Universal Robots PolyScope program: Albert_Miquel.urp

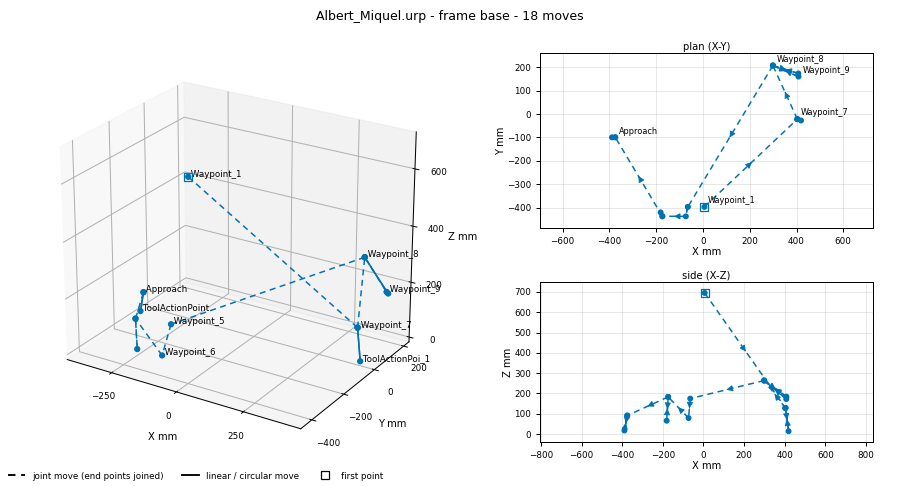
[picture p0: tool path of Albert_Miquel.urp in frame base, 18 of 18 moves have a stored position in this frame; points joined in program order, loops and branches not executed]
Program Albert_Miquel (installation=default directory=/programs createdIn=5.14.5 lastSavedIn=5.14.5 robotSerialNumber=20195300809)
Calibrated DH parameters: a=[-0.000085, -0.20076, -0.212369, 0.000121, -0.000118, 0]; d=[0.15185, -26.306375, 24.753047, 1.684739, 0.085386, 0.092088]; alpha=[1.572149, -0.00522, -0.011864, 1.571339, -1.571085, 0]; deltaTheta=[0, 0.599885, -0.513355, -0.086555, 0.000006, 0]
InitVariablesNode variables(variable(name=Pallet_1_cnt_1, expression=1), variable(name=Pallet_1_cnt_2, expression=1), variable(name=Pallet_1_lct_1, expression=1), variable(name=Pallet_1_lct_2, expression=1), variable(name=Pallet_1_lno_1, expression=1), variable(name=Pallet_1_lno_2, expression=1), variable(name=Pallet_1_sep_1, expression=False), variable(name=Pallet_1_sep_2, expression=False), variable(name=Pallet_1_tct_1, expression=1), variable(name=Pallet_1_tct_2, expression=1))
BeforeStart
  pregunta := True
  URCap Gripper (Robotiq_Grippers, Robotiq Inc.) dataModel(position=0.0, force=70.0, speed=0.0, positionInDouble=0.0, forceInDouble=70.0, speedInDouble=0.0, slaveIds=[9], blocking=true)
  cont := 0
Robot Program (runOnlyOnce=false)
  MoveJ speed 60 deg/s, acceleration 80 deg/s^2 (useActiveTCP=true) feature=Base
    Waypoint Waypoint_1: TCP in base x=6.311 y=-396.732 z=694.709 mm, rx=-0.0176 ry=2.2163 rz=-2.2227 rad; joints [-0.354, -90.143, -0.087, -90.442, -0.008, 0.331] deg; TCP offset x=0 y=0 z=174 mm, rx=0 ry=0 rz=0 rad
  MoveJ speed 60 deg/s, acceleration 80 deg/s^2 (useActiveTCP=true) feature=Base
    Waypoint Waypoint_7: TCP in base x=403.616 y=-21.755 z=128.516 mm, rx=2.2302 ry=-2.181 rz=0.0652 rad; joints [17.471, -109.042, -67.217, -93.701, 86.636, 16.615] deg
  URCap Palletizing (polyscope-pallet-impl, Universal Robots) dataModel(palletFeature=Base, isPalletizing=true, Length(key=objectHeight value=0.01 unit=M), Variable(key=referencePoint, variable(featureName=referencePoin_1)), Variable(key=separatorPoint, variable(featureName=separatorPoin_1)), Variable(key=name, variable(name=Pallet_2)), Variable(key=globalCountingVariable, variable(name=Pallet_1_cnt_1, initializeExpression=1)), Variable(key=layerCountingVariable, variable(name=Pallet_1_lct_1, initializeExpression=1)), Variable(key=layerNumberVariable, variable(name=Pallet_1_lno_1, initializeExpression=1)), Variable(key=handleSeparatorVariable, variable(name=Pallet_1_sep_1, initializeExpression=False)), Variable(key=totalCountVariable, variable(name=Pallet_1_tct_1, initializeExpression=1))); state(isChildrenLocked=true)
    URCap Patterns (polyscope-pallet-impl, Universal Robots) state(isChildrenLocked=true)
      URCap Pattern (polyscope-pallet-impl, Universal Robots) dataModel(UUID=8c053362-77a5-4536-95ea-2a82096237cb, patternType=GRID, rows=2, columns=3, Variable(key=nameVariable, variable(name=Grid_Pattern_2))); state(isChildrenLocked=true)
        URCap Item (polyscope-pallet-impl, Universal Robots) dataModel(UUID=2fe570d1-5f2a-4909-ad3f-dfae3d26dd40, patternType=GRID, index=0, calibrationDeltaTheta=[2.0871938292282843E-8, 0.5998849625986696, -0.513354759222901, -0.08655474087847535, 6.239817607139875E-6, -6.658617090343766E-8], calibrationA=[-8.52060452638757E-5, -0.2007601879611388, -0.2123691625519033, 1.2105607098011576E-4, -1.1833705743435544E-4, 0.0], calibrationD=[0.15184970286177432, -26.306374840159272, 24.75304670983349, 1.6847390881089916, 0.085385969004481, 0.09208826337351553], calibrationAlpha=[1.5721487795181908, -0.005219907129425837, -0.011864150755780208, 1.5713392161993658, -1.5710853432049288, 0.0], calibrationJointChecksum=[-1860213401, -1859864814, -1494669377, -1328152407, -1329437658, -1329056899], calibrationStatus=2, calibrationValidChecksum=true, baseToFeature=[0.0, 0.0, 0.0, 0.0, 0.0, 0.0], TCPOffset=[-1.4423623202718117E-5, -9.352838594822721E-6, 0.17400406362699186, 1.4244432014475435E-5, 1.820526178641711E-5, -5.9448890467481114E-5], Variable(key=variable, variable(name=CornerItem_5)), JointPositions(key=jointpositions, JointPosition(key=[1], Angle(key=pos value=0.250581 unit=RAD)), JointPosition(key=[2], Angle(key=pos value=-2.028934 unit=RAD)), JointPosition(key=[3], Angle(key=pos value=-1.566597 unit=RAD)), JointPosition(key=[4], Angle(key=pos value=-1.060673 unit=RAD)), JointPosition(key=[5], Angle(key=pos value=1.557171 unit=RAD)), JointPosition(key=[6], Angle(key=pos value=0.245986 unit=RAD))))
        URCap Item (polyscope-pallet-impl, Universal Robots) dataModel(UUID=48b683ab-8145-4bec-8b11-a3f435976ee8, patternType=GRID, index=1, calibrationDeltaTheta=[2.0871938292282843E-8, 0.5998849625986696, -0.513354759222901, -0.08655474087847535, 6.239817607139875E-6, -6.658617090343766E-8], calibrationA=[-8.52060452638757E-5, -0.2007601879611388, -0.2123691625519033, 1.2105607098011576E-4, -1.1833705743435544E-4, 0.0], calibrationD=[0.15184970286177432, -26.306374840159272, 24.75304670983349, 1.6847390881089916, 0.085385969004481, 0.09208826337351553], calibrationAlpha=[1.5721487795181908, -0.005219907129425837, -0.011864150755780208, 1.5713392161993658, -1.5710853432049288, 0.0], calibrationJointChecksum=[-1860213401, -1859864814, -1494669377, -1328152407, -1329437658, -1329056899], calibrationStatus=2, calibrationValidChecksum=true, baseToFeature=[0.0, 0.0, 0.0, 0.0, 0.0, 0.0], TCPOffset=[-1.4207780571977302E-5, 1.2223832136171175E-5, 0.1740135199298931, -3.519253042201217E-5, 1.1066226283473242E-5, -7.594307323318983E-5], Variable(key=variable, variable(name=CornerItem_6)), JointPositions(key=jointpositions, JointPosition(key=[1], Angle(key=pos value=0.345107 unit=RAD)), JointPosition(key=[2], Angle(key=pos value=-1.682404 unit=RAD)), JointPosition(key=[3], Angle(key=pos value=-1.989274 unit=RAD)), JointPosition(key=[4], Angle(key=pos value=-1.065282 unit=RAD)), JointPosition(key=[5], Angle(key=pos value=1.556964 unit=RAD)), JointPosition(key=[6], Angle(key=pos value=0.300862 unit=RAD))))
        URCap Item (polyscope-pallet-impl, Universal Robots) dataModel(UUID=2ec47bc2-6cf6-4d25-ba3f-7980db0fa51f, patternType=GRID, index=2, calibrationDeltaTheta=[2.0871938292282843E-8, 0.5998849625986696, -0.513354759222901, -0.08655474087847535, 6.239817607139875E-6, -6.658617090343766E-8], calibrationA=[-8.52060452638757E-5, -0.2007601879611388, -0.2123691625519033, 1.2105607098011576E-4, -1.1833705743435544E-4, 0.0], calibrationD=[0.15184970286177432, -26.306374840159272, 24.75304670983349, 1.6847390881089916, 0.085385969004481, 0.09208826337351553], calibrationAlpha=[1.5721487795181908, -0.005219907129425837, -0.011864150755780208, 1.5713392161993658, -1.5710853432049288, 0.0], calibrationJointChecksum=[-1860213401, -1859864814, -1494669377, -1328152407, -1329437658, -1329056899], calibrationStatus=2, calibrationValidChecksum=true, baseToFeature=[0.0, 0.0, 0.0, 0.0, 0.0, 0.0], TCPOffset=[2.5368332041697528E-6, -7.638363482442845E-6, 0.1739966047788814, 2.5498434355735236E-5, 1.9165595671850262E-5, -4.160228463273833E-7], Variable(key=variable, variable(name=CornerItem_7)), JointPositions(key=jointpositions, JointPosition(key=[1], Angle(key=pos value=-0.292791 unit=RAD)), JointPosition(key=[2], Angle(key=pos value=-1.985792 unit=RAD)), JointPosition(key=[3], Angle(key=pos value=-1.581072 unit=RAD)), JointPosition(key=[4], Angle(key=pos value=-1.161729 unit=RAD)), JointPosition(key=[5], Angle(key=pos value=1.568378 unit=RAD)), JointPosition(key=[6], Angle(key=pos value=-0.312319 unit=RAD))))
        URCap Item (polyscope-pallet-impl, Universal Robots) dataModel(UUID=376d6808-81de-4906-a0ef-a0a6ed99bf62, patternType=GRID, index=3, calibrationDeltaTheta=[2.0871938292282843E-8, 0.5998849625986696, -0.513354759222901, -0.08655474087847535, 6.239817607139875E-6, -6.658617090343766E-8], calibrationA=[-8.52060452638757E-5, -0.2007601879611388, -0.2123691625519033, 1.2105607098011576E-4, -1.1833705743435544E-4, 0.0], calibrationD=[0.15184970286177432, -26.306374840159272, 24.75304670983349, 1.6847390881089916, 0.085385969004481, 0.09208826337351553], calibrationAlpha=[1.5721487795181908, -0.005219907129425837, -0.011864150755780208, 1.5713392161993658, -1.5710853432049288, 0.0], calibrationJointChecksum=[-1860213401, -1859864814, -1494669377, -1328152407, -1329437658, -1329056899], calibrationStatus=2, calibrationValidChecksum=true, baseToFeature=[0.0, 0.0, 0.0, 0.0, 0.0, 0.0], TCPOffset=[2.5499804027467876E-5, -1.257017656741688E-6, 0.17398892781983108, 3.7811907055945986E-5, 4.437019733495021E-5, 8.204365596035897E-6], Variable(key=variable, variable(name=CornerItem_8)), JointPositions(key=jointpositions, JointPosition(key=[1], Angle(key=pos value=-0.223663 unit=RAD)), JointPosition(key=[2], Angle(key=pos value=-2.250266 unit=RAD)), JointPosition(key=[3], Angle(key=pos value=-1.184856 unit=RAD)), JointPosition(key=[4], Angle(key=pos value=-1.225029 unit=RAD)), JointPosition(key=[5], Angle(key=pos value=1.552142 unit=RAD)), JointPosition(key=[6], Angle(key=pos value=-0.257117 unit=RAD))))
    URCap Layers (polyscope-pallet-impl, Universal Robots) dataModel(separators=[false], selectedPatterns=[8c053362-77a5-4536-95ea-2a82096237cb])
    URCap At Each Item (polyscope-pallet-impl, Universal Robots) dataModel(selectedPattern=8c053362-77a5-4536-95ea-2a82096237cb, selectedPosition=2fe570d1-5f2a-4909-ad3f-dfae3d26dd40, Approach_calibrationDeltaTheta=[2.0871938292282843E-8, 0.5998849625986696, -0.513354759222901, -0.08655474087847535, 6.239817607139875E-6, -6.658617090343766E-8], Approach_calibrationA=[-8.52060452638757E-5, -0.2007601879611388, -0.2123691625519033, 1.2105607098011576E-4, -1.1833705743435544E-4, 0.0], Approach_calibrationD=[0.15184970286177432, -26.306374840159272, 24.75304670983349, 1.6847390881089916, 0.085385969004481, 0.09208826337351553], Approach_calibrationAlpha=[1.5721487795181908, -0.005219907129425837, -0.011864150755780208, 1.5713392161993658, -1.5710853432049288, 0.0], Approach_calibrationJointChecksum=[-1860213401, -1859864814, -1494669377, -1328152407, -1329437658, -1329056899], Approach_calibrationStatus=2, Approach_calibrationValidChecksum=true, Approach_baseToFeature=[0.0, 0.0, 0.0, 0.0, 0.0, 0.0], Approach_TCPOffset=[-1.9077118991468744E-5, 4.457855078521256E-6, 0.17399737117322073, 3.6181022651684704E-6, -2.272290840480485E-5, -2.3439487455844403E-5], Exit_calibrationDeltaTheta=[2.0871938292282843E-8, 0.5998849625986696, -0.513354759222901, -0.08655474087847535, 6.239817607139875E-6, -6.658617090343766E-8], Exit_calibrationA=[-8.52060452638757E-5, -0.2007601879611388, -0.2123691625519033, 1.2105607098011576E-4, -1.1833705743435544E-4, 0.0], Exit_calibrationD=[0.15184970286177432, -26.306374840159272, 24.75304670983349, 1.6847390881089916, 0.085385969004481, 0.09208826337351553], Exit_calibrationAlpha=[1.5721487795181908, -0.005219907129425837, -0.011864150755780208, 1.5713392161993658, -1.5710853432049288, 0.0], Exit_calibrationJointChecksum=[-1860213401, -1859864814, -1494669377, -1328152407, -1329437658, -1329056899], Exit_calibrationStatus=2, Exit_calibrationValidChecksum=true, Exit_baseToFeature=[0.0, 0.0, 0.0, 0.0, 0.0, 0.0], Exit_TCPOffset=[-5.374249363220007E-6, -2.3174252664071027E-6, 0.1739743665157666, 4.7864739912950294E-5, -1.859553978069823E-5, -2.935668304045453E-5], currentWizardState=LANDING, Pose(key=refBaseToFeature, Position(key=posePosition, Length(key=X value=0 unit=M), Length(key=Y value=0 unit=M), Length(key=Z value=0 unit=M)), Rotation(key=poseRotation, Angle(key=RX value=0 unit=RAD), Angle(key=RY value=0 unit=RAD), Angle(key=RZ value=0 unit=RAD))), Pose(key=refPose, Position(key=posePosition, Length(key=X value=0.421311 unit=M), Length(key=Y value=-0.018191 unit=M), Length(key=Z value=0.010406 unit=M)), Rotation(key=poseRotation, Angle(key=RX value=2.240112 unit=RAD), Angle(key=RY value=-2.177821 unit=RAD), Angle(key=RZ value=0.113453 unit=RAD))), JointPositions(key=Approach_jointpositions, JointPosition(key=[1], Angle(key=pos value=0.304932 unit=RAD)), JointPosition(key=[2], Angle(key=pos value=-1.90314 unit=RAD)), JointPosition(key=[3], Angle(key=pos value=-1.173158 unit=RAD)), JointPosition(key=[4], Angle(key=pos value=-1.635384 unit=RAD)), JointPosition(key=[5], Angle(key=pos value=1.512082 unit=RAD)), JointPosition(key=[6], Angle(key=pos value=0.289982 unit=RAD))), JointPositions(key=Exit_jointpositions, JointPosition(key=[1], Angle(key=pos value=0.304932 unit=RAD)), JointPosition(key=[2], Angle(key=pos value=-1.90314 unit=RAD)), JointPosition(key=[3], Angle(key=pos value=-1.173158 unit=RAD)), JointPosition(key=[4], Angle(key=pos value=-1.635384 unit=RAD)), JointPosition(key=[5], Angle(key=pos value=1.512082 unit=RAD)), JointPosition(key=[6], Angle(key=pos value=0.289982 unit=RAD))))
      URCap Generated Movements (polyscope-pallet-impl, Universal Robots) state(isChildrenLocked=true)
        MoveJ speed 60 deg/s, acceleration 80 deg/s^2 (useActiveTCP=true) feature=referencePoin_1
          Waypoint Approach_1: TCP in base x=403.611 y=-21.736 z=128.518 mm, rx=2.2302 ry=-2.181 rz=0.0652 rad; joints [17.471, -109.042, -67.217, -93.701, 86.636, 16.615] deg; TCP offset x=-0.019 y=0.004 z=173.997 mm, rx=0 ry=0 rz=0 rad; feature pose in base x=421.311 y=-18.191 z=10.406 mm, rx=2.2401 ry=-2.1778 rz=0.1135 rad
        MoveL speed 250 mm/s, acceleration 1200 mm/s^2 (useActiveTCP=true) feature(featureName=referencePoin_1)
          Waypoint ToolActionPoi_1: TCP in base x=419.174 y=-27.418 z=14.219 mm, rx=-2.1938 ry=2.1821 rz=-0.0468 rad; joints [14.357, -116.249, -89.759, -60.772, 89.219, 14.094] deg; TCP offset x=0 y=0 z=174 mm, rx=0 ry=0 rz=0 rad
        Folder Tool action
          URCap Gripper (Robotiq_Grippers, Robotiq Inc.) dataModel(position=88.62745098039215, force=96.0, speed=0.0, positionInDouble=88.62745098039215, forceInDouble=96.0, speedInDouble=0.0, slaveIds=[9], blocking=true)
        MoveL speed 250 mm/s, acceleration 1200 mm/s^2 (useActiveTCP=true) feature(featureName=referencePoin_1)
          Waypoint Exit_2: TCP in base x=403.618 y=-21.748 z=128.541 mm, rx=2.2303 ry=-2.181 rz=0.0652 rad; joints [17.471, -109.042, -67.217, -93.701, 86.636, 16.615] deg; TCP offset x=-0.005 y=-0.002 z=173.974 mm, rx=0 ry=0 rz=0 rad
  cont := cont+1
  If cont≟2
    MoveJ speed 60 deg/s, acceleration 80 deg/s^2 (useActiveTCP=true) feature=Base
      Waypoint Waypoint_8: TCP in base x=298.99 y=207.505 z=263.54 mm, rx=-3.0265 ry=-0.0112 rz=-0.0377 rad; joints [-171.587, -73.732, 33.631, -52.328, -84.428, -81.357] deg; TCP offset x=0 y=0 z=174 mm, rx=0 ry=0 rz=0 rad
    MoveJ speed 60 deg/s, acceleration 80 deg/s^2 (useActiveTCP=true) feature=Base
      Waypoint Waypoint_9: TCP in base x=408.571 y=160.257 z=184.062 mm, rx=3.127 ry=-0.0032 rz=0.1029 rad; joints [-175.411, -60.326, 38.564, -71.943, -91.9, -85.088] deg
    URCap Gripper (Robotiq_Grippers, Robotiq Inc.) dataModel(position=0.0, force=85.0, speed=0.0, positionInDouble=0.0, forceInDouble=85.0, speedInDouble=0.0, slaveIds=[9], blocking=true)
    MoveJ speed 60 deg/s, acceleration 80 deg/s^2 (useActiveTCP=true) feature=Base
      Waypoint Waypoint_10: TCP in base x=298.999 y=207.517 z=263.537 mm, rx=-3.0265 ry=-0.0112 rz=-0.0377 rad; joints [-171.587, -73.731, 33.632, -52.33, -84.427, -81.358] deg
    pregunta :=  (valueSource=Operator message=buena? valueType=Boolean)
    cont := 0
    If pregunta≟ False
      Wait Sleep waitTime=1
    Else 
      MoveJ speed 60 deg/s, acceleration 80 deg/s^2 (useActiveTCP=true) feature=Base
        Waypoint Waypoint_11: TCP in base x=407.765 y=173.494 z=172.615 mm, rx=-3.1188 ry=-0.0111 rz=-0.0636 rad; joints [-174.935, -59.077, 39.218, -72.594, -89.797, -85.087] deg
      URCap Gripper (Robotiq_Grippers, Robotiq Inc.) dataModel(position=100.0, force=85.0, speed=0.0, positionInDouble=100.0, forceInDouble=85.0, speedInDouble=0.0, slaveIds=[9], blocking=true)
      MoveJ speed 60 deg/s, acceleration 80 deg/s^2 (useActiveTCP=true) feature=Base
        Waypoint Waypoint_12: TCP in base x=299 y=207.509 z=263.546 mm, rx=-3.0265 ry=-0.0113 rz=-0.0377 rad; joints [-171.588, -73.732, 33.631, -52.33, -84.427, -81.362] deg
  Else 
    Wait Sleep waitTime=1
  If pregunta≟ True
    MoveJ speed 60 deg/s, acceleration 80 deg/s^2 (useActiveTCP=true) feature=Base
      Waypoint Waypoint_5: TCP in base x=-64.631 y=-396.801 z=174.762 mm, rx=0.0621 ry=3.0949 rz=0.0444 rad; joints [-82.48, -115.107, -45.299, -110.777, 92.204, 10.413] deg
    MoveJ speed 60 deg/s, acceleration 80 deg/s^2 (useActiveTCP=true) feature=Base
      Waypoint Waypoint_6: TCP in base x=-73.197 y=-437.247 z=79.067 mm, rx=2.2405 ry=-2.1614 rz=-0.0322 rad; joints [-81.257, -120.175, -64.027, -85.752, 87.254, -82.979] deg
      URCap Gripper (Robotiq_Grippers, Robotiq Inc.) dataModel(position=0.0, force=85.0, speed=0.0, positionInDouble=0.0, forceInDouble=85.0, speedInDouble=0.0, slaveIds=[9], blocking=true)
  Else 
    pregunta := True
  If digital_in[0]≟ False
    MoveJ speed 60 deg/s, acceleration 80 deg/s^2 (useActiveTCP=true) feature=Base
      Waypoint Waypoint_2: TCP in base x=-173.442 y=-436.915 z=182.927 mm, rx=2.1717 ry=-2.1648 rz=0.004 rad; joints [52.337, -47.529, 16.835, -63.608, -91.247, -127.592] deg
    MoveJ speed 60 deg/s, acceleration 80 deg/s^2 (useActiveTCP=true) feature=Base
      Waypoint Waypoint_3: TCP in base x=-180.921 y=-420.236 z=65.874 mm, rx=-2.1893 ry=2.2229 rz=0.016 rad; joints [50.259, -52.928, 56.702, -92.501, -91.339, -128.883] deg
    URCap Gripper (Robotiq_Grippers, Robotiq Inc.) dataModel(position=100.0, force=85.0, speed=0.0, positionInDouble=100.0, forceInDouble=85.0, speedInDouble=0.0, slaveIds=[9], blocking=true)
    MoveJ speed 60 deg/s, acceleration 80 deg/s^2 (useActiveTCP=true) feature=Base
      Waypoint Waypoint_4: TCP in base x=-173.451 y=-436.914 z=182.947 mm, rx=2.1717 ry=-2.1648 rz=0.004 rad; joints [52.336, -47.531, 16.835, -63.609, -91.248, -127.592] deg
    URCap Palletizing (polyscope-pallet-impl, Universal Robots) dataModel(palletFeature=Base, isPalletizing=true, Length(key=objectHeight value=0.01 unit=M), Variable(key=referencePoint, variable(featureName=referencePoint)), Variable(key=separatorPoint, variable(featureName=separatorPoint)), Variable(key=name, variable(name=Pallet_3)), Variable(key=globalCountingVariable, variable(name=Pallet_1_cnt_2, initializeExpression=1)), Variable(key=layerCountingVariable, variable(name=Pallet_1_lct_2, initializeExpression=1)), Variable(key=layerNumberVariable, variable(name=Pallet_1_lno_2, initializeExpression=1)), Variable(key=handleSeparatorVariable, variable(name=Pallet_1_sep_2, initializeExpression=False)), Variable(key=totalCountVariable, variable(name=Pallet_1_tct_2, initializeExpression=1))); state(isChildrenLocked=true)
      URCap Patterns (polyscope-pallet-impl, Universal Robots) state(isChildrenLocked=true)
        URCap Pattern (polyscope-pallet-impl, Universal Robots) dataModel(UUID=8c053362-77a5-4536-95ea-2a82096237cb, patternType=GRID, columns=3, rows=2, Variable(key=nameVariable, variable(name=Grid_Pattern_3))); state(isChildrenLocked=true)
          URCap Item (polyscope-pallet-impl, Universal Robots) dataModel(UUID=2fe570d1-5f2a-4909-ad3f-dfae3d26dd40, patternType=GRID, index=0, calibrationDeltaTheta=[2.0871938292282843E-8, 0.5998849625986696, -0.513354759222901, -0.08655474087847535, 6.239817607139875E-6, -6.658617090343766E-8], calibrationA=[-8.52060452638757E-5, -0.2007601879611388, -0.2123691625519033, 1.2105607098011576E-4, -1.1833705743435544E-4, 0.0], calibrationD=[0.15184970286177432, -26.306374840159272, 24.75304670983349, 1.6847390881089916, 0.085385969004481, 0.09208826337351553], calibrationAlpha=[1.5721487795181908, -0.005219907129425837, -0.011864150755780208, 1.5713392161993658, -1.5710853432049288, 0.0], calibrationJointChecksum=[-1860213401, -1859864814, -1494669377, -1328152407, -1329437658, -1329056899], calibrationStatus=2, calibrationValidChecksum=true, baseToFeature=[0.0, 0.0, 0.0, 0.0, 0.0, 0.0], TCPOffset=[1.2287880736761014E-5, 1.4603764760257043E-6, 0.1739907052327735, 8.925285764918683E-6, 3.273907169153255E-5, 4.254307635580523E-5], Variable(key=variable, variable(name=CornerItem_9)), JointPositions(key=jointpositions, JointPosition(key=[1], Angle(key=pos value=-0.092053 unit=RAD)), JointPosition(key=[2], Angle(key=pos value=-1.158893 unit=RAD)), JointPosition(key=[3], Angle(key=pos value=1.614853 unit=RAD)), JointPosition(key=[4], Angle(key=pos value=-2.039518 unit=RAD)), JointPosition(key=[5], Angle(key=pos value=-1.572956 unit=RAD)), JointPosition(key=[6], Angle(key=pos value=-0.112591 unit=RAD))))
          URCap Item (polyscope-pallet-impl, Universal Robots) dataModel(UUID=48b683ab-8145-4bec-8b11-a3f435976ee8, patternType=GRID, index=1, calibrationDeltaTheta=[2.0871938292282843E-8, 0.5998849625986696, -0.513354759222901, -0.08655474087847535, 6.239817607139875E-6, -6.658617090343766E-8], calibrationA=[-8.52060452638757E-5, -0.2007601879611388, -0.2123691625519033, 1.2105607098011576E-4, -1.1833705743435544E-4, 0.0], calibrationD=[0.15184970286177432, -26.306374840159272, 24.75304670983349, 1.6847390881089916, 0.085385969004481, 0.09208826337351553], calibrationAlpha=[1.5721487795181908, -0.005219907129425837, -0.011864150755780208, 1.5713392161993658, -1.5710853432049288, 0.0], calibrationJointChecksum=[-1860213401, -1859864814, -1494669377, -1328152407, -1329437658, -1329056899], calibrationStatus=2, calibrationValidChecksum=true, baseToFeature=[0.0, 0.0, 0.0, 0.0, 0.0, 0.0], TCPOffset=[3.972253346168353E-6, -1.0811753194950313E-6, 0.17397580939523236, 1.3771020395959111E-5, 2.3380738252636774E-5, 9.263728897875755E-6], Variable(key=variable, variable(name=CornerItem_10)), JointPositions(key=jointpositions, JointPosition(key=[1], Angle(key=pos value=-0.072467 unit=RAD)), JointPosition(key=[2], Angle(key=pos value=-0.775889 unit=RAD)), JointPosition(key=[3], Angle(key=pos value=0.981079 unit=RAD)), JointPosition(key=[4], Angle(key=pos value=-1.808238 unit=RAD)), JointPosition(key=[5], Angle(key=pos value=-1.560334 unit=RAD)), JointPosition(key=[6], Angle(key=pos value=-0.090196 unit=RAD))))
          URCap Item (polyscope-pallet-impl, Universal Robots) dataModel(UUID=2ec47bc2-6cf6-4d25-ba3f-7980db0fa51f, patternType=GRID, index=2, calibrationDeltaTheta=[2.0871938292282843E-8, 0.5998849625986696, -0.513354759222901, -0.08655474087847535, 6.239817607139875E-6, -6.658617090343766E-8], calibrationA=[-8.52060452638757E-5, -0.2007601879611388, -0.2123691625519033, 1.2105607098011576E-4, -1.1833705743435544E-4, 0.0], calibrationD=[0.15184970286177432, -26.306374840159272, 24.75304670983349, 1.6847390881089916, 0.085385969004481, 0.09208826337351553], calibrationAlpha=[1.5721487795181908, -0.005219907129425837, -0.011864150755780208, 1.5713392161993658, -1.5710853432049288, 0.0], calibrationJointChecksum=[-1860213401, -1859864814, -1494669377, -1328152407, -1329437658, -1329056899], calibrationStatus=2, calibrationValidChecksum=true, baseToFeature=[0.0, 0.0, 0.0, 0.0, 0.0, 0.0], TCPOffset=[1.5475995746028204E-5, -1.430186872564132E-5, 0.1739931236891783, 1.7143936766620148E-5, -5.3348595293828974E-6, 1.4419079550804771E-5], Variable(key=variable, variable(name=CornerItem_11)), JointPositions(key=jointpositions, JointPosition(key=[1], Angle(key=pos value=0.315313 unit=RAD)), JointPosition(key=[2], Angle(key=pos value=-0.521391 unit=RAD)), JointPosition(key=[3], Angle(key=pos value=0.546652 unit=RAD)), JointPosition(key=[4], Angle(key=pos value=-1.716915 unit=RAD)), JointPosition(key=[5], Angle(key=pos value=-1.575083 unit=RAD)), JointPosition(key=[6], Angle(key=pos value=0.31151 unit=RAD))))
          URCap Item (polyscope-pallet-impl, Universal Robots) dataModel(UUID=376d6808-81de-4906-a0ef-a0a6ed99bf62, patternType=GRID, index=3, calibrationDeltaTheta=[2.0871938292282843E-8, 0.5998849625986696, -0.513354759222901, -0.08655474087847535, 6.239817607139875E-6, -6.658617090343766E-8], calibrationA=[-8.52060452638757E-5, -0.2007601879611388, -0.2123691625519033, 1.2105607098011576E-4, -1.1833705743435544E-4, 0.0], calibrationD=[0.15184970286177432, -26.306374840159272, 24.75304670983349, 1.6847390881089916, 0.085385969004481, 0.09208826337351553], calibrationAlpha=[1.5721487795181908, -0.005219907129425837, -0.011864150755780208, 1.5713392161993658, -1.5710853432049288, 0.0], calibrationJointChecksum=[-1860213401, -1859864814, -1494669377, -1328152407, -1329437658, -1329056899], calibrationStatus=2, calibrationValidChecksum=true, baseToFeature=[0.0, 0.0, 0.0, 0.0, 0.0, 0.0], TCPOffset=[8.16938922265642E-6, -7.364140791388252E-6, 0.17401649354888465, -2.3147522346839827E-5, 8.331106328931583E-6, 1.6576102854599155E-5], JointPositions(key=jointpositions, JointPosition(key=[1], Angle(key=pos value=0.459706 unit=RAD)), JointPosition(key=[2], Angle(key=pos value=-0.798006 unit=RAD)), JointPosition(key=[3], Angle(key=pos value=1.012531 unit=RAD)), JointPosition(key=[4], Angle(key=pos value=-1.772857 unit=RAD)), JointPosition(key=[5], Angle(key=pos value=-1.689658 unit=RAD)), JointPosition(key=[6], Angle(key=pos value=0.43449 unit=RAD))), Variable(key=variable, variable(name=CornerItem_12)))
      URCap Layers (polyscope-pallet-impl, Universal Robots) dataModel(separators=[false], selectedPatterns=[8c053362-77a5-4536-95ea-2a82096237cb])
      URCap At Each Item (polyscope-pallet-impl, Universal Robots) dataModel(currentWizardState=MANUAL, selectedPattern=8c053362-77a5-4536-95ea-2a82096237cb, selectedPosition=2fe570d1-5f2a-4909-ad3f-dfae3d26dd40, Pose(key=refBaseToFeature, Position(key=posePosition, Length(key=X value=0 unit=M), Length(key=Y value=0 unit=M), Length(key=Z value=0 unit=M)), Rotation(key=poseRotation, Angle(key=RX value=0 unit=RAD), Angle(key=RY value=0 unit=RAD), Angle(key=RZ value=0 unit=RAD))), Pose(key=refPose, Position(key=posePosition, Length(key=X value=-0.413059 unit=M), Length(key=Y value=-0.104843 unit=M), Length(key=Z value=0.02231 unit=M)), Rotation(key=poseRotation, Angle(key=RX value=-2.227947 unit=RAD), Angle(key=RY value=-2.152214 unit=RAD), Angle(key=RZ value=-0.072993 unit=RAD))))
        URCap Generated Movements (polyscope-pallet-impl, Universal Robots) state(isChildrenLocked=true)
          MoveJ speed 60 deg/s, acceleration 80 deg/s^2 (useActiveTCP=true) feature=referencePoint
            Waypoint Approach: TCP in base x=-374.933 y=-99.241 z=91.188 mm, rx=-2.1869 ry=-2.1814 rz=-0.069 rad; joints [-2.271, -72.738, 80.807, -98.535, -94.72, -2.147] deg; feature pose in base x=-413.059 y=-104.843 z=22.31 mm, rx=-2.2279 ry=-2.1522 rz=-0.073 rad
          MoveL speed 250 mm/s, acceleration 1200 mm/s^2 (useActiveTCP=true) feature(featureName=referencePoint)
            Waypoint ToolActionPoint: TCP in base x=-388.778 y=-99.414 z=17.541 mm, rx=-2.2012 ry=-2.2376 rz=0.0257 rad; joints [-5.277, -66.401, 92.524, -116.853, -90.126, -6.448] deg
          Folder Tool action
            URCap Gripper (Robotiq_Grippers, Robotiq Inc.) dataModel(position=0.0, force=0.0, speed=0.0, positionInDouble=0.0, forceInDouble=0.0, speedInDouble=0.0, slaveIds=[9], blocking=true)
          MoveL speed 250 mm/s, acceleration 1200 mm/s^2 (useActiveTCP=true) feature(featureName=referencePoint)
            Waypoint Exit_1: TCP in base x=-374.923 y=-99.233 z=91.151 mm, rx=-2.187 ry=-2.1814 rz=-0.069 rad; joints [-2.275, -72.735, 80.81, -98.536, -94.717, -2.15] deg
Thread Thread_1 (runOnlyOnce=false)
  If digital_in[0]≟ False
    Set DigitalOutput pin=digital_out[0]; digitalValue=0
  Else 
    Set DigitalOutput pin=digital_out[0]; digitalValue=1
